// TIA Portal V17 export
// export: Created 2021-12-03T08:12:54.7408227Z, ExportSetting WithDefaults, DisplayName Totally Integrated Automation Portal, DisplayVersion V17, DisplayName TIA Portal Openness, DisplayVersion V17, DisplayName TIA Portal Version Control Interface, DisplayVersion V17, DisplayName STEP 7 Professional, DisplayVersion V17, DisplayName STEP 7 Safety, DisplayVersion V17, DisplayName WinCC Advanced, DisplayVersion V17
FUNCTION_BLOCK "FB_DetLineCtrl"   // FB21, FBD
VERSION : 0.1
// stored: AutoNumber false, IsIECCheckEnabled false, UDAEnableTagReadback false
   VAR_INPUT
      ID : Int;
      LADDR : Word;
      I_StartScan : Bool;
      I_StopScan : Bool;
      I_Setup : Bool;
      I_Speed : Int;
      I_Direct : Bool;
      I_HighDose : Bool;
   END_VAR
   VAR DB_SPECIFIC
      Telegr : Struct
         MsgID : DWord;
         MsgLen : DWord;
         ScanData : DWord;
         VehSpd : DWord;
      END_STRUCT;
      TCP_Sts : Struct
         Done : Bool;
         Error : Bool;
         Status : Word;
         Len : Int;
         ErrCd : Word;
      END_STRUCT;
      StrtTelegr : Bool;
      StrtTelegr_His : Bool;
      StrtTelegrSts : Bool;
      StrtTelegrSts_His : Bool;
   END_VAR
   VAR_TEMP   // added for the SCL form of the ladder/FBD networks
      _w1 : Bool;
      _w2 : Bool;
   END_VAR
BEGIN

REGION Network 1
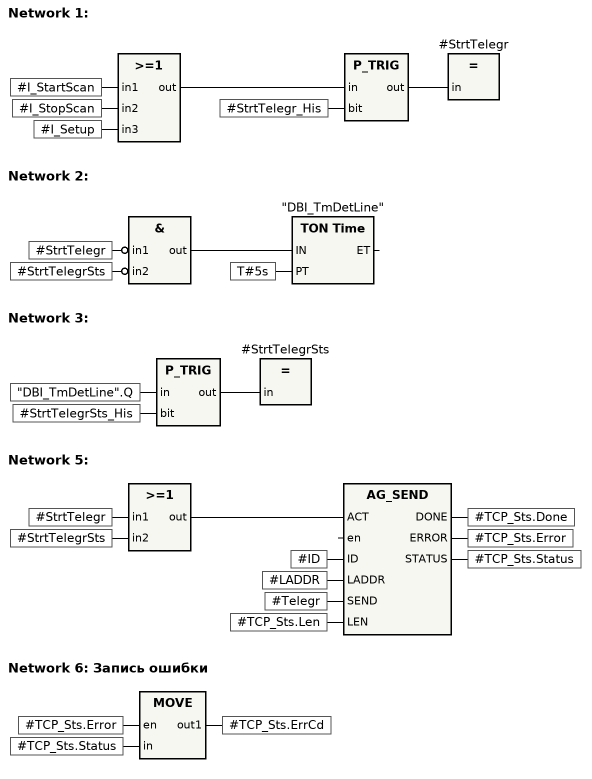
   #_w1 := #I_StartScan OR #I_StopScan OR #I_Setup;
   #_w2 := #_w1 AND NOT #StrtTelegr_His;   // rising edge
   #StrtTelegr_His := #_w1;
   #StrtTelegr := #_w2;
END_REGION

REGION Network 2
   "DBI_TmDetLine".TON(IN := NOT #StrtTelegr AND NOT #StrtTelegrSts, PT := T#5s);
END_REGION

REGION Network 3
   #_w1 := "DBI_TmDetLine".Q AND NOT #StrtTelegrSts_His;   // rising edge
   #StrtTelegrSts_His := "DBI_TmDetLine".Q;
   #StrtTelegrSts := #_w1;
END_REGION

NETWORK
TITLE = 
      A     #I_StartScan;
      JCN   Strt;

      L     1;
      T     #Telegr.MsgID;
Strt: NOP   0;

      A     #I_StopScan;
      JCN   Stp;

      L     2;
      T     #Telegr.MsgID;
Stp:  NOP   0;

      A     #I_Setup;
      JCN   Setup;

      L     3;
      T     #Telegr.MsgID;
Setup:NOP   0;

      L     16;
      T     #Telegr.MsgLen;

      L     16;
      T     #TCP_Sts.Len;

      A     #StrtTelegrSts;
      JCN   Sts;

      L     0;
      T     #Telegr.MsgID;

      L     8;
      T     #Telegr.MsgLen;

      L     8;
      T     #TCP_Sts.Len;
Sts:  NOP   0;



      L     #I_Speed;
      T     #Telegr.VehSpd;

      A     #I_HighDose;
      =     "DetLineSnd_HighDose";
      A     #I_Direct;
      =     "DetLineSnd_Direct";
      L     "DetLineSnd_ScanData";
      CAW;
      T     #Telegr.ScanData;

REGION Network 5
   AG_SEND(ACT := #StrtTelegr OR #StrtTelegrSts,
           ID := #ID,
           LADDR := #LADDR,
           SEND := #Telegr,
           LEN := #TCP_Sts.Len,
           DONE => #TCP_Sts.Done,
           ERROR => #TCP_Sts.Error,
           STATUS => #TCP_Sts.Status);
END_REGION

REGION Network 6: Запись ошибки
   IF #TCP_Sts.Error THEN #TCP_Sts.ErrCd := #TCP_Sts.Status; END_IF;
END_REGION
END_FUNCTION_BLOCK
